// Mitsubishi GX Works2 project: 0625(카운트2)   PLC: Q02/Q02H

PROGRAM MAIN
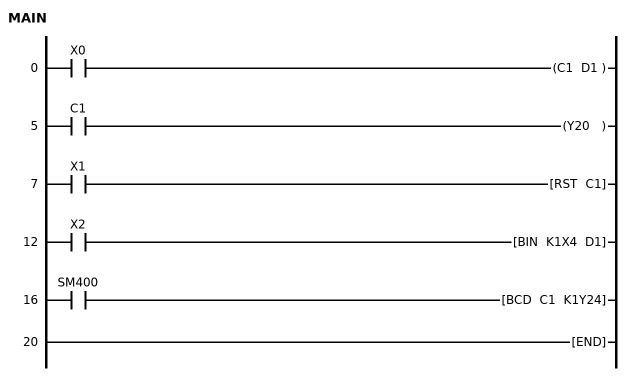
0     LD      X0
      OUT     C1 D1
5     LD      C1
      OUT     Y20
7     LD      X1
      RST     C1
12    LD      X2
      BIN     K1X4 D1
16    LD      SM400
      BCD     C1 K1Y24
20    END
END_PROGRAM
